// TIA Portal V20 export
TYPE "typeUnitMode"
// stored: Access Published, IsFailsafeCompliant true, Namespace Safety
   STRUCT
      production : Bool;
      maintanance : Bool;
      manual : Bool;
      noMode : Bool;
   END_STRUCT;
END_TYPE
